FUNCTION Convert_USINT_TO_LREAL : Hresult
VAR_INPUT
	in : USINT;
	out : REFERENCE TO LREAL;
END_VAR
VAR
	converted : LREAL;
END_VAR
VAR CONSTANT
	INCOMPATIBLE : HRESULT := 16#9811070E;
END_VAR

converted := USINT_TO_LREAL(in);

IF (LREAL_TO_USINT(converted) <> in) THEN
	Convert_USINT_TO_LREAL := INCOMPATIBLE;
	RETURN;
END_IF

out := converted;

END_FUNCTION

(* stored: Version 1.1.0.1, ProductVersion 3.1.4024.12
   POU Convert_USINT_TO_LREAL: Id {e67dcd7b-2a9e-4b32-8fb7-6a57214deb81}, SpecialFunc None *)
